FUNCTION_BLOCK Fb_FeederOperation
VAR_INPUT
	nModeSelector	: FeederMode;
	bEnable         : BOOL;
END_VAR
VAR_OUTPUT
	bJogFwd         : BOOL;
	bJogRev         : BOOL;
END_VAR
VAR
END_VAR

;

END_FUNCTION_BLOCK

(* stored: Version 1.1.0.1, ProductVersion 3.1.4024.12
   POU Fb_FeederOperation: Id {cda18660-b2b1-423c-9389-c10dbb890a58}, SpecialFunc None *)
